{attribute 'qualified_only'}
{attribute 'strict'}
TYPE SafeState :
(
	Init := 0,
	Close,
	CheckDigit,
	Open,
	WrongCode
);
END_TYPE

(* stored: Version 1.1.0.1, ProductVersion 3.1.4024.13
   DUT SafeState: Id {ed3dc943-1481-41e6-8463-b12791cdc564} *)
